# EPICS SNL sequencer program: seq/test/validate/userfunc.st
/*************************************************************************\
Copyright (c) 2010-2012 Helmholtz-Zentrum Berlin f. Materialien
                        und Energie GmbH, Germany (HZB)
This file is distributed subject to a Software License Agreement found
in the file LICENSE that is included with this distribution.
\*************************************************************************/
program userfuncTest

%%#include "../testSupport.h"

option +s;

%{
static void incr(SS_ID ssId, int *pv, VAR_ID v)
{
    seq_pvGet(ssId, v, SYNC);
    *pv += 1;
    seq_pvPut(ssId, v, SYNC);
}
}%

int i = 0;
assign i;
monitor i;

foreign pVar, ssId;

entry {
    seq_test_init(10);
}

ss myss {
    state doit {
        int i_saved;
        when (delay(0.1)) {
            incr(ssId, &i, pvIndex(i));
            testOk1(i_saved == i-1);
            i_saved = i;
        } state doit
        when (i == 10) {
        } exit
    }
}

exit {
    seq_test_done();
}
